{attribute 'qualified_only'}
{attribute 'strict'}
TYPE E_SourceType : 
(
	eLive := 0,
	eHistMQTT,
	eHistFile
) ;
END_TYPE

(* stored: DUT E_SourceType: Id 170b8cc2-e491-4f86-841f-3815ae5a0c15 *)
